# B&R Automation Studio project Sim_task1_plc
Automation Studio 4.5.2.102; Simulerings opgave 1 - PLC del

## Configuration Config1

### Hardware
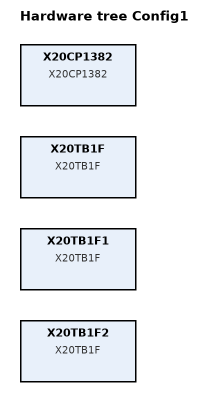
```
X20CP1382 : X20CP1382 v1.7.0.0  [X1 -> X1.SL; X2 -> X2.SL; X3 -> X3.SL]
  Module X1 (Type=X1, Virtual=true, Version=1.7.0.0)
    Connection (Connector=SS1, TargetModule=X20TB1F, TargetConnector=SS)
    Connection (Connector=SL, TargetModule=X20CP1382, TargetConnector=X1)
  Module X2 (Type=X2, Virtual=true, Version=1.7.0.0)
    Connection (Connector=SS1, TargetModule=X20TB1F1, TargetConnector=SS)
    Connection (Connector=SL, TargetModule=X20CP1382, TargetConnector=X2)
  Module X3 (Type=X3, Virtual=true, Version=1.7.0.0)
    Connection (Connector=SS1, TargetModule=X20TB1F2, TargetConnector=SS)
    Connection (Connector=SL, TargetModule=X20CP1382, TargetConnector=X3)
  Connector IF2:
    ActivateDevice = 1
  ConfigurationID = Sim_task1_plc_Config1
X20TB1F : X20TB1F v1.0.0.0
X20TB1F1 : X20TB1F v1.0.0.0
X20TB1F2 : X20TB1F v1.0.0.0
```

## Logical view

### Types.typ - Local data types
```iecst
TYPE
	box : 	STRUCT
		lenght : UINT;
		type : Box_type;
		width : UINT;
		area : UINT;
	END_STRUCT;
	Box_type :
		(
		sml,
		lrg,
		med
		);
	operation :
		(
		meassuring,
		calculation,
		waiting
		);
END_TYPE
```

### shared_vars.var
```iecst
VAR
	next_box : box;
END_VAR
```

### Program Logical/Sorting_programs/meassure (IEC)

#### Main.st - Init, cyclic, exit code
```iecst
PROGRAM _INIT
	 STATE := waiting;
END_PROGRAM

PROGRAM _CYCLIC
	//state logic
	CASE STATE OF
		waiting:
			IF di_laser1 THEN
				STATE := meassuring;
			END_IF

		meassuring:
			IF NOT di_laser1 THEN
				STATE := calculation;
			END_IF

		calculation:

	END_CASE

	//state I/O
	CASE STATE OF
		meassuring:
			laser_timer.IN := TRUE;
			laser_timer.PT := T#2000ms;
			laser_timer();
			IF di_laser1 THEN
				current_box.width := BELT_WIDTH - ai_laser1;
			END_IF

		calculation:
			current_box.lenght := TIME_TO_UINT (laser_timer.ET);
			current_box.area := current_box.lenght * 2 + current_box.width * 2;
			IF current_box.area < 800 THEN
				current_box.type := sml;
			ELSIF current_box.area < 1000 THEN
				current_box.type := med;
			ELSE
				current_box.type := lrg;
			END_IF

			next_box := current_box;

			laser_timer.IN := FALSE;
			laser_timer();
			STATE := waiting;

	END_CASE

END_PROGRAM

PROGRAM _EXIT
	(* Insert code here *)

END_PROGRAM
```

#### Variables.var - Local variables
```iecst
VAR CONSTANT
	BELT_SPEED : UINT := 1000;
	BELT_WIDTH : UINT := 650;
	FIXED_HEIGHT : UINT := 0;
END_VAR
VAR
	ai_laser1 : UINT;
	laser_timer : TON;
	STATE : operation;
	current_box : box;
	di_laser1 : BOOL;
END_VAR
```

### Program Logical/Sorting_programs/sort_V2 (IEC)

#### Variables.var
```iecst
VAR
	do_pusher2 : BOOL;
	do_pusher1 : BOOL;
	timer : TON;
	di_laser4 : BOOL;
	push_timer : TON;
END_VAR
```

#### Main.st
```iecst
PROGRAM _INIT

END_PROGRAM

PROGRAM _CYCLIC
	CASE next_box.type OF
		sml:
			IF di_laser4 THEN
				timer.PT := T#350ms;
				timer.IN := TRUE;
			END_IF
			IF timer.Q THEN
				timer.IN := FALSE;
				timer();
				//push
				push_timer.IN := TRUE;
				push_timer.PT := T#400ms;
				push_timer();
				do_pusher1 := TRUE;
			END_IF
			IF push_timer.Q THEN
				do_pusher1 := FALSE;
				push_timer.IN := FALSE;
			END_IF
		med:
			IF di_laser4 THEN
				timer.PT := T#1250ms;
				timer.IN := TRUE;
			END_IF
			IF timer.Q THEN
				timer.IN := FALSE;
				timer();
				//push
				push_timer.IN := TRUE;
				push_timer.PT := T#400ms;
				push_timer();
				do_pusher2 := TRUE;
			END_IF
			IF push_timer.Q THEN
				do_pusher2 := FALSE;
				push_timer.IN := FALSE;
			END_IF
	END_CASE

	timer();
	push_timer();
END_PROGRAM

PROGRAM _EXIT

END_PROGRAM
```

### Program Logical/Sorting_programs/sort (IEC)

#### Variables.var
```iecst
VAR
	di_laser2 : BOOL;
	di_laser3 : BOOL;
	do_pusher2 : BOOL;
	do_pusher1 : BOOL;
	trigger : F_TRIG;
	push_timer : TON;
END_VAR
```

#### Main.st
```iecst
PROGRAM _INIT
	push_timer.PT := T#300ms;

END_PROGRAM

PROGRAM _CYCLIC
	CASE next_box.type OF
		sml:
			trigger.CLK := di_laser2;
			trigger();
			IF trigger.Q THEN
				do_pusher1 :=  NOT push_timer.Q;
				push_timer.IN := TRUE;
				push_timer();
			END_IF
			IF NOT push_timer.Q THEN
				do_pusher1 := FALSE;
				push_timer.IN := FALSE;
				push_timer();
			END_IF

		med:
			trigger.CLK := di_laser3;
			do_pusher2 := NOT push_timer.Q;
			trigger();
			IF trigger.Q THEN
				push_timer.IN := TRUE;
				push_timer();
			END_IF
			(*IF NOT push_timer.Q THEN
				push_timer.IN := FALSE;
				push_timer();
			END_IF*)

		lrg:
			//DAB
			do_pusher1 := FALSE;
			do_pusher2 := FALSE;
	END_CASE

END_PROGRAM

PROGRAM _EXIT
	(* Insert code here *)

END_PROGRAM
```

### Program Logical/meassure

#### Variables.var
```iecst
VAR CONSTANT
	BELT_SPEED : UINT := 1000;
	BELT_WIDTH : UINT := 650;
	FIXED_HEIGHT : UINT := 0;
END_VAR
VAR
	di_laser1 : BOOL;
	ai_laser1 : UINT;
	laser_timer : TON;
	STATE : operation;
	current_box : box;
END_VAR
```

#### Main.st
```iecst
PROGRAM _INIT
	 STATE := waiting;
END_PROGRAM

PROGRAM _CYCLIC
	//state logic
	CASE STATE OF
		waiting:
			IF di_laser1 THEN
				STATE := meassuring;
			END_IF

		meassuring:
			IF NOT di_laser1 THEN
				STATE := calculation;
			END_IF

		calculation:

	END_CASE

	//state I/O
	CASE STATE OF
		meassuring:
			laser_timer.IN := TRUE;
			laser_timer.PT := T#2000ms;
			laser_timer();
			IF di_laser1 THEN
				current_box.width := BELT_WIDTH - ai_laser1;
			END_IF

		calculation:
			current_box.lenght := TIME_TO_UINT (laser_timer.ET);
			current_box.area := current_box.lenght * 2 + current_box.width * 2;
			IF current_box.area < 633 THEN
				current_box.type := sml;
			ELSIF current_box.area < 866 THEN
				current_box.type := med;
			ELSE
				current_box.type := lrg;
			END_IF

			laser_timer.IN := FALSE;
			STATE := waiting;

	END_CASE

END_PROGRAM

PROGRAM _EXIT
	(* Insert code here *)

END_PROGRAM
```

Listed in the project but not available here: Logical/Global.typ, Logical/Global.var, Logical/Libraries
